// TIA Portal project "Project1" (V17)

(* hardware
DEVICE "S7-1200 station_1"  S7-1200 Station
   slot 0: "Rack_0"  S7-1200 Rack  Rack  V1.0
   slot 1: "PLC_1"  CPU 1214C AC/DC/Rly  6ES7 214-1BE30-0XB0  V2.2
*)

// ===== PLC "PLC_1"  CPU 1214C AC/DC/Rly =====

VAR_GLOBAL   // PLC tag table "Default tag table"
   "entrada" AT %M100.0 : Bool;
   "salida" AT %M100.1 : Bool;
   "Tag_1" AT %MW200 : Word;
   "verde" AT %M100.2 : Bool;
   "ambar" AT %M100.3 : Bool;
   "rojo" AT %M100.4 : Bool;
   "Tag_2" AT %MW300 : Int;
   "Tag_3" AT %M400.1 : Bool;
   "Tag_4" AT %M400.2 : Bool;
END_VAR

DATA_BLOCK "Data_block_1"   // DB1
{ S7_Optimized_Access := 'TRUE' }
VERSION : 0.1
BEGIN
END_DATA_BLOCK

DATA_BLOCK "Block_1_DB"   // DB3
{ S7_Optimized_Access := 'TRUE' }
VERSION : 0.1
// stored: InstanceOfName Block_1
"Block_1"
BEGIN
END_DATA_BLOCK

// folder: System blocks/Program resources

DATA_BLOCK "IEC_Counter_0_DB"   // DB2
{ S7_Optimized_Access := 'TRUE' }
AUTHOR : Simatic
FAMILY : IEC
NAME : CNTR
VERSION : 1.0
// stored: InstanceOfName IEC_COUNTER
"IEC_COUNTER"
BEGIN
END_DATA_BLOCK

// folder: (top level)

FUNCTION_BLOCK "Block_1"   // FB1, LAD
{ S7_Optimized_Access := 'TRUE' }
VERSION : 0.1
// Se va a crear un garaje automático gestionado por un PLC, y se montará la información en un Dashboard creado con NodeRed y la informacion del garaje se guardara en una base de datos local que utilizaremos MySQL. Es decir, conectarenos otro servidor a NodeRed
BEGIN

REGION Network 1
   // El bloque CTUD es un contador y es el que se encarga de contar y descontar los automoviles que entran.
   // CU: cuenta los coches que entran 
   // CD:dectecta los coches que salen y los resata de la base de datos 
   // R:resetea 
   // LD:cagar los valores del contador 
   // PV: es el limite 
   // CV: se guardan los datos del contador
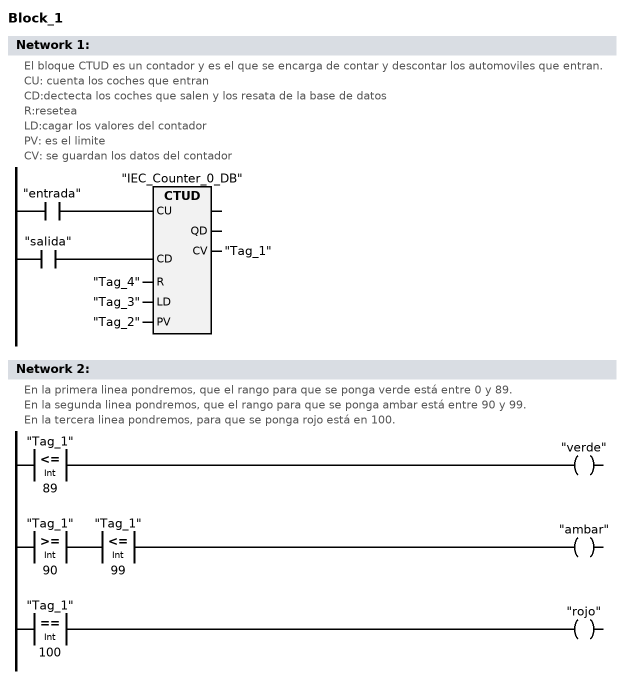
   "IEC_Counter_0_DB".CTUD(CU := "entrada",
                           CD := "salida",
                           R := "Tag_4",
                           LD := "Tag_3",
                           PV := "Tag_2",
                           CV => "Tag_1");
END_REGION

REGION Network 2
   // En la primera linea pondremos, que el rango para que se ponga verde está entre 0 y 89.
   // En la segunda linea pondremos, que el rango para que se ponga ambar está entre 90 y 99.
   // En la tercera linea pondremos, para que se ponga rojo está en 100.
   RUNG wire#powerrail
      { S7_Templates := "SrcType := Int" } LE_Contact(in1 := "Tag_1", in2 := 89)
      Coil( "verde" )
   END_RUNG
   RUNG wire#powerrail
      { S7_Templates := "SrcType := Int" } GE_Contact(in1 := "Tag_1", in2 := 90)
      { S7_Templates := "SrcType := Int" } LE_Contact(in1 := "Tag_1", in2 := 99)
      Coil( "ambar" )
   END_RUNG
   RUNG wire#powerrail
      { S7_Templates := "SrcType := Int" } EQ_Contact(in1 := "Tag_1", in2 := 100)
      Coil( "rojo" )
   END_RUNG
   // the same network as SCL:
   "verde" := "Tag_1" <= 89;
   "ambar" := ("Tag_1" >= 90) AND ("Tag_1" <= 99);
   "rojo" := "Tag_1" = 100;
END_REGION
END_FUNCTION_BLOCK

ORGANIZATION_BLOCK "Main"   // OB1, LAD, ProgramCycle
TITLE = "Main Program Sweep (Cycle)"
{ S7_Optimized_Access := 'TRUE' }
VERSION : 0.1
BEGIN

REGION Network 1
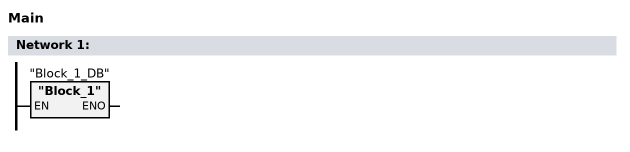
   RUNG wire#powerrail
      "Block_1_DB"()
   END_RUNG
   // the same network as SCL:
   "Block_1_DB"();   // "Block_1"
END_REGION
END_ORGANIZATION_BLOCK